// TIA Portal V21 export
VAR_GLOBAL   // PLC tag table "KAllSens"
END_VAR
VAR_GLOBAL CONSTANT   // user constants
   KAllSens_Spare : Int := 1;
END_VAR
